% RSLogix 500 project PROJECT1.RSS, saved by version 8.30.00.16 %
PROJECT "PROJECT1"    % processor: Bul.1763 MicroLogix 1100 Series B %

PROGRAM FILES
  LAD 2   22 rungs

DATA FILES
  O0 OUTPUT  5 elements
  I1 INPUT  7 elements
  S2 STATUS  66 elements
  B3 BINARY  3 elements
  T4 TIMER  3 elements
  C5 COUNTER  1 elements
  R6 CONTROL  1 elements
  N7 INTEGER  1 elements
  F8 FLOAT  1 elements

LADDER 2
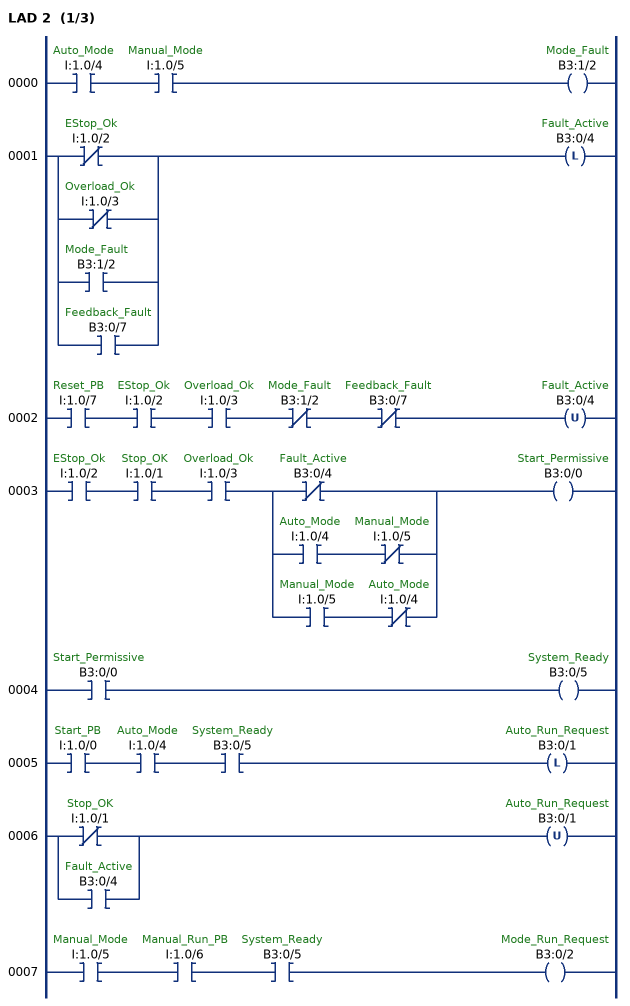
% Rung: 0 %
SOR XIC I:1.0/4 XIC I:1.0/5 OTE B3:1/2 EOR
%   I:1.0/4  "Auto_Mode" %
%   I:1.0/5  "Manual_Mode" %
%   B3:1/2  "Mode_Fault" %
% Rung: 1 %
SOR BST XIO I:1.0/2 NXB BST XIO I:1.0/3 NXB BST XIC B3:1/2 NXB XIC B3:0/7 BND BND BND OTL B3:0/4 EOR
%   I:1.0/2  "EStop_Ok" %
%   I:1.0/3  "Overload_Ok" %
%   B3:1/2  "Mode_Fault" %
%   B3:0/7  "Feedback_Fault" %
%   B3:0/4  "Fault_Active" %
% Rung: 2 %
SOR XIC I:1.0/7 XIC I:1.0/2 XIC I:1.0/3 XIO B3:1/2 XIO B3:0/7 OTU B3:0/4 EOR
%   I:1.0/7  "Reset_PB" %
%   I:1.0/2  "EStop_Ok" %
%   I:1.0/3  "Overload_Ok" %
%   B3:1/2  "Mode_Fault" %
%   B3:0/7  "Feedback_Fault" %
%   B3:0/4  "Fault_Active" %
% Rung: 3 %
SOR XIC I:1.0/2 XIC I:1.0/1 XIC I:1.0/3 BST XIO B3:0/4 NXB BST XIC I:1.0/4 XIO I:1.0/5 NXB XIC I:1.0/5 XIO I:1.0/4 BND BND OTE B3:0/0 EOR
%   I:1.0/2  "EStop_Ok" %
%   I:1.0/1  "Stop_OK" %
%   I:1.0/3  "Overload_Ok" %
%   B3:0/4  "Fault_Active" %
%   I:1.0/4  "Auto_Mode" %
%   I:1.0/5  "Manual_Mode" %
%   B3:0/0  "Start_Permissive" %
% Rung: 4 %
SOR XIC B3:0/0 OTE B3:0/5 EOR
%   B3:0/0  "Start_Permissive" %
%   B3:0/5  "System_Ready" %
% Rung: 5 %
SOR XIC I:1.0/0 XIC I:1.0/4 XIC B3:0/5 OTL B3:0/1 EOR
%   I:1.0/0  "Start_PB" %
%   I:1.0/4  "Auto_Mode" %
%   B3:0/5  "System_Ready" %
%   B3:0/1  "Auto_Run_Request" %
% Rung: 6 %
SOR BST XIO I:1.0/1 NXB XIC B3:0/4 BND OTU B3:0/1 EOR
%   I:1.0/1  "Stop_OK" %
%   B3:0/4  "Fault_Active" %
%   B3:0/1  "Auto_Run_Request" %
% Rung: 7 %
SOR XIC I:1.0/5 XIC I:1.0/6 XIC B3:0/5 OTE B3:0/2 EOR
%   I:1.0/5  "Manual_Mode" %
%   I:1.0/6  "Manual_Run_PB" %
%   B3:0/5  "System_Ready" %
%   B3:0/2  "Mode_Run_Request" %

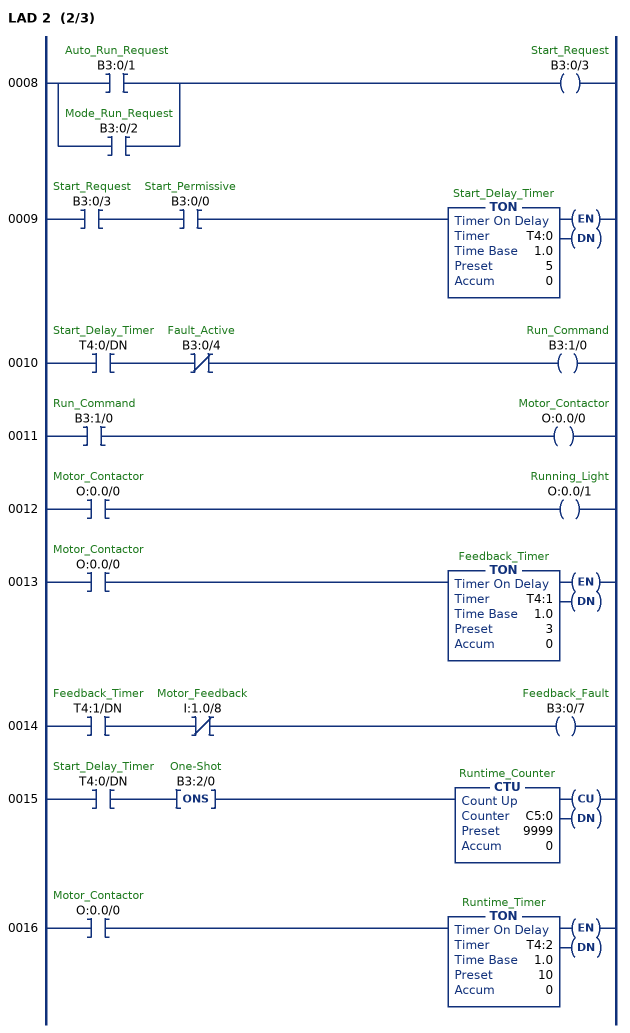
% Rung: 8 %
SOR BST XIC B3:0/1 NXB XIC B3:0/2 BND OTE B3:0/3 EOR
%   B3:0/1  "Auto_Run_Request" %
%   B3:0/2  "Mode_Run_Request" %
%   B3:0/3  "Start_Request" %
% Rung: 9 %
SOR XIC B3:0/3 XIC B3:0/0 TON T4:0 1.0 5 0 EOR
%   B3:0/3  "Start_Request" %
%   B3:0/0  "Start_Permissive" %
%   T4:0  "Start_Delay_Timer" %
% Rung: 10 %
SOR XIC T4:0/DN XIO B3:0/4 OTE B3:1/0 EOR
%   T4:0  "Start_Delay_Timer" %
%   B3:0/4  "Fault_Active" %
%   B3:1/0  "Run_Command" %
% Rung: 11 %
SOR XIC B3:1/0 OTE O:0.0/0 EOR
%   B3:1/0  "Run_Command" %
%   O:0.0/0  "Motor_Contactor" %
% Rung: 12 %
SOR XIC O:0.0/0 OTE O:0.0/1 EOR
%   O:0.0/0  "Motor_Contactor" %
%   O:0.0/1  "Running_Light" %
% Rung: 13 %
SOR XIC O:0.0/0 TON T4:1 1.0 3 0 EOR
%   O:0.0/0  "Motor_Contactor" %
%   T4:1  "Feedback_Timer" %
% Rung: 14 %
SOR XIC T4:1/DN XIO I:1.0/8 OTE B3:0/7 EOR
%   T4:1  "Feedback_Timer" %
%   I:1.0/8  "Motor_Feedback" %
%   B3:0/7  "Feedback_Fault" %
% Rung: 15 %
SOR XIC T4:0/DN ONS B3:2/0 CTU C5:0 9999 0 EOR
%   T4:0  "Start_Delay_Timer" %
%   B3:2/0  "One-Shot" %
%   C5:0  "Runtime_Counter" %
% Rung: 16 %
SOR XIC O:0.0/0 TON T4:2 1.0 10 0 EOR
%   O:0.0/0  "Motor_Contactor" %
%   T4:2  "Runtime_Timer" %

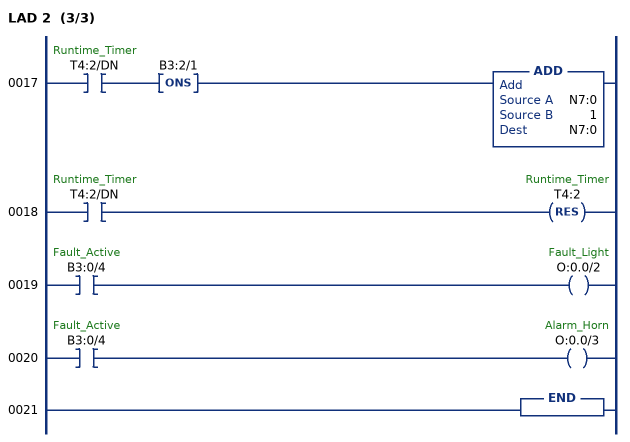
% Rung: 17 %
SOR XIC T4:2/DN ONS B3:2/1 ADD N7:0 1 N7:0 EOR
%   T4:2  "Runtime_Timer" %
% Rung: 18 %
SOR XIC T4:2/DN RES T4:2 EOR
%   T4:2  "Runtime_Timer" %
% Rung: 19 %
SOR XIC B3:0/4 OTE O:0.0/2 EOR
%   B3:0/4  "Fault_Active" %
%   O:0.0/2  "Fault_Light" %
% Rung: 20 %
SOR XIC B3:0/4 OTE O:0.0/3 EOR
%   B3:0/4  "Fault_Active" %
%   O:0.0/3  "Alarm_Horn" %
% Rung: 21 %
SOR END EOR

OTHER DOCUMENTED ADDRESSES
  B3:1/3  "Mode_Fault"
  I:0.0/7  "RESET_PB"
  I:0.0/8  "Motor_Feedback"
  I:1.1/1  "Stop_Ok"

DATA TABLE (non-zero values as saved)
DATA B3
% B3:0 % 0X0021 0X0000 0X0000
DATA T4
% .PRE .ACC %
% T4:0 % 5 0
% T4:1 % 3 0
% T4:2 % 10 0
DATA C5
% .PRE .ACC %
% C5:0 % 9999 0
